// TIA Portal V20 export
DATA_BLOCK "BK21"   // DB249
// stored: MemoryReserve 100
   VAR
      "X10-1.SEPA CLAMP&CUTTER X-AXIS LIMIT SENSOR(-)" : Bool := TRUE;
      "X10-2.SEPA CLAMP&CUTTER X-AXIS HOME SENSOR" : Bool := TRUE;
      "X12-1.SEPA CLAMP&CUTTER X-AXIS LIMIT SENSOR(+)" : Bool := TRUE;
      "X12-2.SPARE" : Bool := FALSE;
      "X14-1.SEPA GRIPPER X-AXIS LIMIT SENSOR(-)" : Bool := TRUE;
      "X14-2.SEPA GRIPPER X-AXIS HOME SENSOR" : Bool := TRUE;
      "X16-1.SEPA GRIPPER X-AXIS LIMIT SENSOR(+)" : Bool := TRUE;
      "X16-2.SPARE" : Bool := FALSE;
   END_VAR
BEGIN
END_DATA_BLOCK
